FUNCTION_BLOCK WcState
VAR
	{attribute addProperty Name  "<#EC Working Counter State (1=Data Invalid)#>"}		
	_WcState AT %I* : BOOL;
	{attribute addProperty Name  "<#EC Togle bit#>"}		
	_InputToggle AT %I* : BOOL;		
END_VAR

END_FUNCTION_BLOCK

(* stored: Version 1.1.0.1, ProductVersion 3.1.4024.6
   POU WcState: Id {3a54e593-f291-46c2-b410-819f7d3b1efa}, SpecialFunc None *)
